FUNCTION F_ToANY : __SYSTEM.AnyType
VAR_INPUT
	Input: ANY;
END_VAR
VAR
END_VAR

F_ToANY:= Input;

END_FUNCTION

(* stored: POU F_ToANY: Id 2675c069-5856-413d-8e3e-223b23172961, SpecialFunc None *)
